SUBAPPLICATION Uebung_020h (* DigitalInput_I1 auf DigitalOutput_Q1; E_PULSE; Impulsformend *)
  (* Standard: 61499-2 *)
  (* Version 1.0, 2023-10-23, franz *)
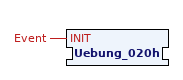
  EVENT_INPUT
    INIT;
  END_EVENT
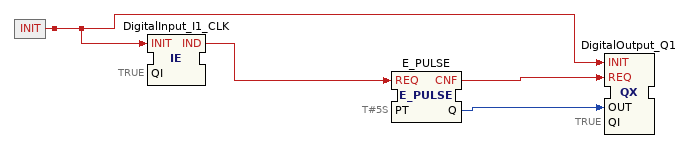
  FBS
    DigitalOutput_Q1 : QX(QI := TRUE);
    E_PULSE : E_PULSE(PT := T#5S);
    DigitalInput_I1_CLK : IE(QI := TRUE);
  END_FBS
  EVENT_CONNECTIONS
    INIT TO DigitalOutput_Q1.INIT;
    E_PULSE.CNF TO DigitalOutput_Q1.REQ;
    DigitalInput_I1_CLK.IND TO E_PULSE.REQ;
    INIT TO DigitalInput_I1_CLK.INIT;
  END_CONNECTIONS
  DATA_CONNECTIONS
    E_PULSE.Q TO DigitalOutput_Q1.OUT;
  END_CONNECTIONS
END_SUBAPPLICATION
